// TIA Portal V20 export
TYPE "UserDiag_typeActIOSystem"
TITLE = UserDiag_typeActIOSystem
   STRUCT
      actIOSystemNumber : Int := 1;   // Number of actual selected IO-system/DP-Mastersystem
      actIODeviceNumbers : Array[1.."USERDIAG_DEVICES_PER_SCREEN_UPPER_LIM"] of UInt;   // Device numbers/profibus addresses of actual selected IO-System/DP-Mastersystem
      actIODeviceState : Array[1.."USERDIAG_DEVICES_PER_SCREEN_UPPER_LIM"] of USInt;   // State of devices/slaves in actual selected IO-System/DP-Mastersystem
      actDeviceSlotsUsed : Array[0.."USERDIAG_SLOTS_PER_SCREEN_UPPER_LIM"] of Bool;   // Used slots of actual selected device/slave
      actDeviceSlotsState : Array[0.."USERDIAG_SLOTS_PER_SCREEN_UPPER_LIM"] of USInt;   // States of actual selected device/slave
   END_STRUCT;
END_TYPE
